// TIA Portal V18 export
// export: Created 2025-12-01T17:52:55.0259752Z, ExportSetting None, DisplayName Totally Integrated Automation Portal, DisplayVersion V18 Update 5, DisplayName TIA Portal Openness, DisplayVersion V18 Update 5, DisplayName TIA Portal Teamcenter Gateway, DisplayVersion V18, DisplayName TIA Portal Version Control Interface, DisplayVersion V18, DisplayName STEP 7 Professional, DisplayVersion V18 Update 5, DisplayName STEP 7 Safety, DisplayVersion V18, DisplayName WinCC Professional, DisplayVersion V18 Update 5
Screen "123ProcessValue1"  1280x800, Number=124, Template=01Auto
  ScreenLayer 
    FaceplateInstance "Process_Data_1" at 10,89 size 425x285  FaceplateTypeName=ProcessData@$@Process_Data V 0.0.13
      Property_1 := AutoProcessData_A_ScanRotate
      InterfacePropertyText "Name_t"  Text="A_ShaftScan / ShaftScan1"
    FaceplateInstance "Process_Data_2" at 430,89 size 425x285  FaceplateTypeName=ProcessData@$@Process_Data V 0.0.13
      Property_1 := AutoProcessData_F_Robot1Grip1
      InterfacePropertyText "Name_t"  Text="F_Robot1Grip1"
    FaceplateInstance "Process_Data_3" at 850,89 size 425x285  FaceplateTypeName=ProcessData@$@Process_Data V 0.0.13
      Property_1 := AutoProcessData_F_Robot1Grip2
      InterfacePropertyText "Name_t"  Text="F_Robot1Grip2"
    FaceplateInstance "Process_Data_4" at 10,388 size 425x285  FaceplateTypeName=ProcessData@$@Process_Data V 0.0.13
      Property_1 := AutoProcessData_B_Press1
      InterfacePropertyText "Name_t"  Text="B_Press1"
    FaceplateInstance "Process_Data_5" at 430,388 size 425x285  FaceplateTypeName=ProcessData@$@Process_Data V 0.0.13
      Property_1 := AutoProcessData_C_Glue
      InterfacePropertyText "Name_t"  Text="C_Glue"
    FaceplateInstance "Process_Data_6" at 850,388 size 425x285  FaceplateTypeName=ProcessData@$@Process_Data V 0.0.13
      Property_1 := AutoProcessData_F_Robot2Grip1
      InterfacePropertyText "Name_t"  Text="F_Robot2Grip1"
    Button "btnMenu6" at 640,725 size 128x75  StyleItem=BtnActive18, TextOff="过程 数据1 / Process Data_1", TextOn="过程 数据1 / Process Data_1"
      on Click: ActivateScreen(Screen name := , Object number := 0); SetTag(Tag := Sys_VersionManagement_HMIPageID, Value := 123)
    Button "btnMenu7_1" at 768,725 size 128x75  StyleItem=BtnNormal20, TextOff="过程 数据2 / Process Data_2", TextOn="过程 数据2 / Process Data_2"
      on Click: ActivateScreen(Screen name := 123ProcessValue2, Object number := 0); SetTag(Tag := Sys_VersionManagement_HMIPageID, Value := 123)
    Button "btnMenu6_2" at 512,725 size 128x75  StyleItem=BtnNormal20, TextOff="工装 扫码数据 / Tooling ScanData / ToolingScan Data", TextOn="工装 扫码数据 / Tooling ScanData / ToolingScan Data"
      on Click: ActivateScreen(Screen name := 125ProcessValue3, Object number := 0); SetTag(Tag := Sys_VersionManagement_HMIPageID, Value := 125)
    Button "btnMenu7_2" at 896,725 size 128x75  StyleItem=BtnNormal20, TextOff="过程 数据Buffer / Process Data_Buffer", TextOn="过程 数据Buffer / Process Data_Buffer"
      on Click: ActivateScreen(Screen name := 129ProcessValue_Buffer, Object number := 0); SetTag(Tag := Sys_VersionManagement_HMIPageID, Value := 129)
    Button "btnMenu7_3" at 1024,725 size 128x75  StyleItem=BtnNormal20, TextOff="过程 数据Buffer / Layout / Process Data_Buffer", TextOn="过程 数据Buffer / Layout / Process Data_Buffer"
      on Click: ActivateScreen(Screen name := 129ProcessValue_Buffer, Object number := 0); SetTag(Tag := Sys_VersionManagement_HMIPageID, Value := 129)
